{attribute 'GeneratedUsingTerminal: AX8108-0100-0101-0101'}
{attribute addProperty BoxType "AX8108-0100-0101-0101"}
{attribute addProperty Id "DeviceMain_OutputsDeviceMain_Outputs_650F34862"}
{attribute addProperty CRC "1847948663"}
{attribute addProperty Size "2"}
TYPE Device_6E257577 :
STRUCT
	{attribute addProperty Name "DeviceMain_Outputs"}
	DeviceMain_Outputs  : DeviceMain_Outputs_650F3486;
END_STRUCT
END_TYPE

(* stored: Version 1.2.0.0, ProductVersion 3.1.4024.11
   DUT Device_6E257577: Id {fad2514b-3c72-4b19-a2c0-fce5666829fe} *)
